(* IEC 61131-3 sources: beckhoffAutomationInterface/ST/Shark/Lib/Communication, 6 files *)

(* ---- GVL_Modbus.st ---- *)
{attribute 'qualified_only'}
(* Modbus protocol constants. *)
VAR_GLOBAL CONSTANT
    MODBUS_MAX_SLAVE_ADDRESS		: BYTE := 247;
    MODBUS_MAX_NETWORK_DEVICES		: BYTE := 8;
    BYTES_PER_REGISTER				: WORD := 2;
    MAX_REGISTERS_PER_OPERATION		: WORD := 32;

    MODBUS_ERROR_INVALID_MASTER		: WORD := 16#8010;
    MODBUS_ERROR_NULL_POINTER		: WORD := 16#8012;
    MODBUS_ERROR_INVALID_QUANTITY	: WORD := 16#8021;
    MODBUS_ERROR_CONVERSION			: WORD := 16#8022;

    MODBUS_DATA_BUFFER_SIZE			: WORD := 64;
    MODBUS_READ_BUFFER_SIZE			: WORD := 32;

    MODBUS_REQUEST_TIMEOUT			: TIME := T#500MS;
END_VAR

(* ---- F_EngineeringToRawCounts.st ---- *)
(* Pure conversion: engineering units to raw Modbus register counts via linear interpolation. *)
FUNCTION F_EngineeringToRawCounts : WORD
VAR_INPUT
    rValue          : LREAL;
    rMinimumValue   : LREAL;
    rFullScale      : LREAL;
    wRawCountsMax   : WORD;
END_VAR
VAR
    rFraction  : LREAL;
    rRawCounts : LREAL;
END_VAR
    IF wRawCountsMax = 0 OR rFullScale <= rMinimumValue THEN
        F_EngineeringToRawCounts := 0;
        RETURN;
    END_IF

    rFraction := (rValue - rMinimumValue) / (rFullScale - rMinimumValue);
    rFraction := LIMIT(0.0, rFraction, 1.0);

    rRawCounts := rFraction * WORD_TO_LREAL(wRawCountsMax);
    F_EngineeringToRawCounts := LREAL_TO_WORD(LIMIT(0.0, rRawCounts, WORD_TO_LREAL(wRawCountsMax)));
END_FUNCTION

(* ---- F_RawCountsToEngineering.st ---- *)
(* Pure conversion: raw Modbus register counts to engineering units via linear interpolation. *)
FUNCTION F_RawCountsToEngineering : LREAL
VAR_INPUT
    wRawCounts      : WORD;
    rMinimumValue   : LREAL;
    rFullScale      : LREAL;
    wRawCountsMax   : WORD;
END_VAR
    IF wRawCountsMax = 0 OR rFullScale <= rMinimumValue THEN
        F_RawCountsToEngineering := 0.0;
        RETURN;
    END_IF

    F_RawCountsToEngineering := rMinimumValue
        + (WORD_TO_LREAL(wRawCounts) / WORD_TO_LREAL(wRawCountsMax))
        * (rFullScale - rMinimumValue);
END_FUNCTION

(* ---- FB_BaseModbusDevice.st ---- *)
(* Base Modbus device handler. Provides FSM for Modbus read/write operations. *)
FUNCTION_BLOCK ABSTRACT FB_BaseModbusDevice IMPLEMENTS I_ModbusSlave
VAR
    _eFSMState 					: E_ModbusDeviceState := E_ModbusDeviceState.IDLE;
    _nUnitId					: BYTE := 0;
    _ipModbusComm				: I_ModbusCommunication := 0;
    _sName						: STRING(80) := 'FB_BaseModbusDevice';
    _fbError					: FB_ErrorHandler;
END_VAR

METHOD PROTECTED SetName
VAR_INPUT
    sName : STRING(80);
END_VAR
    _sName := sName;
    _fbError.Init(sName);
END_METHOD

METHOD PROTECTED RaiseError
VAR_INPUT
    eErrorId : E_ErrorId;
    sMessage : STRING(255);
END_VAR
    _fbError.Raise(eErrorId, sMessage);
END_METHOD

METHOD PROTECTED ClearError
    _fbError.Clear();
END_METHOD

METHOD PUBLIC HandleRequest : BOOL
    IF _eFSMState <> E_ModbusDeviceState.IDLE THEN
        HandleRequest := FALSE;
        RETURN;
    END_IF;

    // NOTE: Do NOT pre-clear the error here. The previous cycle's error stays
    // visible to callers until the next operation actually succeeds, matching
    // the self-healing pattern used by sensors and other controllers.

    // Template-method hook: let the concrete device latch a snapshot of its
    // pending write commands at the start of the transaction. This bounds the
    // write-drain loop even when an upstream controller re-asserts write
    // requests every scan (otherwise the FSM never reaches START_READ/IDLE).
    OnBeginTransaction();

    _eFSMState := E_ModbusDeviceState.START_WRITE;
    HandleRequest := TRUE;
END_METHOD

METHOD PUBLIC Reset : BOOL
    ClearError();
    _eFSMState := E_ModbusDeviceState.IDLE;
    Reset := TRUE;
END_METHOD

METHOD PUBLIC Update : BOOL
    IF _ipModbusComm = 0 THEN
        _eFSMState := E_ModbusDeviceState.IDLE;
        Update := FALSE;
        RETURN;
    END_IF;

    _ipModbusComm.Update();

    CASE _eFSMState OF
        E_ModbusDeviceState.IDLE:
        Update := TRUE;
        RETURN;

        E_ModbusDeviceState.START_WRITE:
        _HandleStartWrite();

        E_ModbusDeviceState.START_READ:
        _HandleStartRead();

        E_ModbusDeviceState.WAIT_FOR_WRITE:
        _HandleWaitForWrite();

        E_ModbusDeviceState.WAIT_FOR_READ:
        _HandleWaitForRead();
    END_CASE;

    Update := TRUE;
END_METHOD

METHOD PRIVATE _HandleStartWrite
VAR
    nWriteStartRegister, nWriteQuantity : WORD;
    pWriteData : POINTER TO BYTE;
END_VAR
    IF GetWritePayload(nStartingRegister => nWriteStartRegister, nQuantity => nWriteQuantity, pData => pWriteData) THEN
        IF _ipModbusComm.StartWriteOperation(nStartRegister := nWriteStartRegister, nQuantity := nWriteQuantity, pData := pWriteData) THEN
            _eFSMState := E_ModbusDeviceState.WAIT_FOR_WRITE;
        END_IF;
    ELSE
        _eFSMState := E_ModbusDeviceState.START_READ;
    END_IF;
END_METHOD

METHOD PRIVATE _HandleStartRead
VAR
    nReadStartRegister, nReadQuantity : WORD;
END_VAR
    IF GetReadPayload(nStartingRegister => nReadStartRegister, nQuantity => nReadQuantity) THEN
        IF _ipModbusComm.StartReadOperation(nStartRegister := nReadStartRegister, nQuantity := nReadQuantity) THEN
            _eFSMState := E_ModbusDeviceState.WAIT_FOR_READ;
        END_IF;
    ELSE
        _eFSMState := E_ModbusDeviceState.IDLE;
    END_IF;
END_METHOD

METHOD PRIVATE _HandleWaitForWrite
VAR
    bSuccess : BOOL;
    wErrorCode : WORD;
END_VAR
    IF NOT _ipModbusComm.IsOperationComplete() THEN
        RETURN;
    END_IF;

    bSuccess := _ipModbusComm.GetOperationResult(wErrorCode);

    IF bSuccess THEN
        ClearError();
        HandleSuccessfulWrite();
    ELSE
        _HandleFailedOperation(wErrorCode);
    END_IF;

    _eFSMState := E_ModbusDeviceState.START_WRITE;
END_METHOD

METHOD PRIVATE _HandleWaitForRead
VAR
    bSuccess : BOOL;
    wErrorCode : WORD;
    pData : POINTER TO BYTE;
    nDataLength : UINT;
END_VAR
    IF NOT _ipModbusComm.IsOperationComplete() THEN
        RETURN;
    END_IF;

    bSuccess := _ipModbusComm.GetOperationResult(wErrorCode);

    IF bSuccess THEN
        ClearError();
        _ipModbusComm.GetReadData(pData, nDataLength);
        HandleSuccessfulRead(pData, nDataLength);
    ELSE
        _HandleFailedOperation(wErrorCode);
    END_IF;

    _eFSMState := E_ModbusDeviceState.IDLE;
END_METHOD

METHOD PRIVATE _HandleFailedOperation
VAR_INPUT
    wErrorCode : WORD;
END_VAR
    RaiseError(E_ErrorId.ERR_COMM_TIMEOUT, CONCAT('Modbus operation failed, code: ', WORD_TO_STRING(wErrorCode)));
END_METHOD

METHOD PUBLIC IsBusy : BOOL
    IsBusy := _eFSMState <> E_ModbusDeviceState.IDLE;
END_METHOD

METHOD PROTECTED _Init : BOOL
VAR_INPUT
    nUnitId						: BYTE;
    ipModbusComm				: I_ModbusCommunication;
END_VAR
    IF ipModbusComm = 0 THEN
        RaiseError(E_ErrorId.ERR_GEN_NULL_POINTER, 'Communication handler is null');
        RETURN;
    END_IF

    _nUnitId := nUnitId;
    _ipModbusComm := ipModbusComm;
    _Init := TRUE;
END_METHOD

METHOD PUBLIC GetUnitId : BYTE
    GetUnitId := _nUnitId;
END_METHOD

METHOD PROTECTED ABSTRACT HandleSuccessfulRead
VAR_INPUT
    pData						: POINTER TO BYTE;
    nDataLength					: UINT;
END_VAR
END_METHOD

METHOD PROTECTED ABSTRACT GetReadPayload : BOOL
VAR_OUTPUT
    nStartingRegister			: WORD;
    nQuantity					: WORD;
END_VAR
END_METHOD

METHOD PROTECTED ABSTRACT GetWritePayload : BOOL
VAR_OUTPUT
    nStartingRegister			: WORD;
    nQuantity					: WORD;
    pData						: POINTER TO BYTE;
END_VAR
END_METHOD

METHOD PROTECTED ABSTRACT HandleSuccessfulWrite
END_METHOD

(* Template-method hook called once at the start of each round-robin transaction
   (IDLE -> START_WRITE). The default implementation is a no-op. Devices whose
   write commands are re-asserted every scan should override this to snapshot the
   pending write requests, so a single transaction stays bounded:
   drain snapshotted writes -> read -> IDLE. *)
METHOD PROTECTED OnBeginTransaction
END_METHOD

END_FUNCTION_BLOCK

(* ---- FB_ModbusHardwareHandler.st ---- *)
(* Modbus hardware communication handler. Wraps Beckhoff ModbusRtuMasterV2_KL6x22B. *)
FUNCTION_BLOCK FB_ModbusHardwareHandler IMPLEMENTS I_ModbusCommunication
VAR
    _fbError            : FB_ErrorHandler;
    _pModbusMaster      : POINTER TO ModbusRtuMasterV2_KL6x22B;
    _nSlaveAddress      : BYTE;
    _bOperationComplete : BOOL := FALSE;
    _wError             : WORD := 0;
    _aDataBuffer        : ARRAY[0..GVL_Modbus.MODBUS_DATA_BUFFER_SIZE-1] OF BYTE;
    _aReadBuffer        : ARRAY[0..GVL_Modbus.MODBUS_READ_BUFFER_SIZE-1] OF WORD;
    _nLastQuantity      : WORD;
    _nLastRegister      : WORD;
    _eLastOperation     : E_ModbusOperationType := E_ModbusOperationType.NONE;
    _bExecuteFlag       : BOOL := FALSE;
END_VAR

METHOD PRIVATE ConvertModbusBytesToWords : BOOL
VAR_INPUT
    pByteData : POINTER TO BYTE;
    nByteCount : WORD;
    pWordBuffer : POINTER TO WORD;
    nMaxWords : WORD;
END_VAR
VAR
    nWordsToConvert : WORD;
END_VAR
    IF pByteData = 0 THEN
        RETURN;
    END_IF

    IF pWordBuffer = 0 THEN
        RETURN;
    END_IF

    IF nByteCount = 0 THEN
        RETURN;
    END_IF

    IF (nByteCount MOD GVL_Modbus.BYTES_PER_REGISTER) <> 0 THEN
        RETURN;
    END_IF

    nWordsToConvert := nByteCount / GVL_Modbus.BYTES_PER_REGISTER;
    IF nWordsToConvert > nMaxWords THEN
        nWordsToConvert := nMaxWords;
    END_IF

    // Bulk copy — data is already in native (little-endian) byte order
    MEMCPY(pWordBuffer, pByteData, nWordsToConvert * SIZEOF(WORD));

    ConvertModbusBytesToWords := TRUE;
END_METHOD

METHOD PRIVATE _ValidateForOperation : BOOL
VAR_INPUT
    nQuantity : WORD;
END_VAR
    IF _pModbusMaster = 0 THEN
        _wError := GVL_Modbus.MODBUS_ERROR_INVALID_MASTER;
        _fbError.Raise(eErrorId := E_ErrorId.ERR_GEN_NULL_POINTER, sMessage := 'Modbus master not initialized');
        RETURN;
    END_IF

    IF _pModbusMaster^.BUSY THEN
        RETURN;
    END_IF

    IF nQuantity = 0 OR nQuantity > GVL_Modbus.MAX_REGISTERS_PER_OPERATION THEN
        _wError := GVL_Modbus.MODBUS_ERROR_INVALID_QUANTITY;
        _fbError.Raise(eErrorId := E_ErrorId.ERR_GEN_INVALID_PARAM, sMessage := 'Invalid register quantity');
        RETURN;
    END_IF

    _ValidateForOperation := TRUE;
END_METHOD

METHOD PUBLIC Init : BOOL
VAR_INPUT
    sInstanceName    : STRING(80);
    pModbusRtuMaster : POINTER TO ModbusRtuMasterV2_KL6x22B;
    nSlaveAddress    : BYTE;
END_VAR
    _fbError.Init(sSourceName := sInstanceName);

    _pModbusMaster := pModbusRtuMaster;
    _nSlaveAddress := nSlaveAddress;

    IF pModbusRtuMaster = 0 THEN
        _fbError.Raise(eErrorId := E_ErrorId.ERR_GEN_NULL_POINTER, sMessage := 'Modbus master pointer is null');
        Init := FALSE;
    ELSE
        _fbError.Clear();
        Init := TRUE;
    END_IF
END_METHOD

METHOD PUBLIC StartReadOperation : BOOL
VAR_INPUT
    nStartRegister : WORD;
    nQuantity : WORD;
END_VAR
    IF NOT _ValidateForOperation(nQuantity := nQuantity) THEN
        RETURN;
    END_IF

    _nLastQuantity := nQuantity;
    _nLastRegister := nStartRegister;
    _eLastOperation := E_ModbusOperationType.READ;
    _bOperationComplete := FALSE;
    _wError := 0;
    _bExecuteFlag := TRUE;
    _fbError.Clear();

    StartReadOperation := TRUE;
END_METHOD

METHOD PUBLIC StartWriteOperation : BOOL
VAR_INPUT
    nStartRegister : WORD;
    nQuantity : WORD;
    pData : POINTER TO BYTE;
END_VAR
    IF NOT _ValidateForOperation(nQuantity := nQuantity) THEN
        RETURN;
    END_IF

    IF pData = 0 THEN
        _wError := GVL_Modbus.MODBUS_ERROR_NULL_POINTER;
        _fbError.Raise(eErrorId := E_ErrorId.ERR_GEN_NULL_POINTER, sMessage := 'Data pointer is null');
        RETURN;
    END_IF

    // Bulk copy — native byte order is little-endian, matching Modbus register layout
    MEMCPY(ADR(_aDataBuffer), pData, nQuantity * GVL_Modbus.BYTES_PER_REGISTER);

    _nLastQuantity := nQuantity;
    _nLastRegister := nStartRegister;
    _eLastOperation := E_ModbusOperationType.WRITE;
    _bOperationComplete := FALSE;
    _wError := 0;
    _bExecuteFlag := TRUE;
    _fbError.Clear();

    StartWriteOperation := TRUE;
END_METHOD

METHOD PUBLIC Update : BOOL
    IF _pModbusMaster = 0 THEN
        _bOperationComplete := TRUE;
        _wError := GVL_Modbus.MODBUS_ERROR_INVALID_MASTER;
        _fbError.Raise(eErrorId := E_ErrorId.ERR_GEN_NULL_POINTER, sMessage := 'Modbus master not initialized');
        Update := TRUE;
        RETURN;
    END_IF

    IF _eLastOperation = E_ModbusOperationType.NONE THEN
        Update := _bOperationComplete;
        RETURN;
    END_IF

    _CallMaster();

    IF NOT _bOperationComplete AND_THEN NOT _pModbusMaster^.BUSY THEN
        _bOperationComplete := TRUE;
        _HandleCompletion();
        _eLastOperation := E_ModbusOperationType.NONE;
    END_IF

    Update := _bOperationComplete;
END_METHOD

METHOD PRIVATE _CallMaster
VAR
    nByteLength : WORD;
END_VAR
    nByteLength := _nLastQuantity * GVL_Modbus.BYTES_PER_REGISTER;

    IF _eLastOperation = E_ModbusOperationType.READ THEN
        _pModbusMaster^.ReadRegs(
            UnitID := _nSlaveAddress,
            Quantity := _nLastQuantity,
            MBAddr := _nLastRegister,
            cbLength := nByteLength,
            pMemoryAddr := ADR(_aDataBuffer),
            Execute := _bExecuteFlag,
            Timeout := GVL_Modbus.MODBUS_REQUEST_TIMEOUT
        );
    ELSIF _eLastOperation = E_ModbusOperationType.WRITE THEN
        _pModbusMaster^.WriteRegs(
            UnitID := _nSlaveAddress,
            Quantity := _nLastQuantity,
            MBAddr := _nLastRegister,
            cbLength := nByteLength,
            pMemoryAddr := ADR(_aDataBuffer),
            Execute := _bExecuteFlag,
            Timeout := GVL_Modbus.MODBUS_REQUEST_TIMEOUT
        );
    END_IF

    _bExecuteFlag := FALSE;
END_METHOD

METHOD PRIVATE _HandleCompletion
VAR
    nActualBytes : WORD;
END_VAR
    IF _pModbusMaster^.Error THEN
        _wError := INT_TO_WORD(_pModbusMaster^.ErrorId);
        _fbError.Raise(eErrorId := E_ErrorId.ERR_COMM_PROTOCOL,
            sMessage := CONCAT('Modbus error code: ', WORD_TO_STRING(_wError)));
        RETURN;
    END_IF

    IF _eLastOperation <> E_ModbusOperationType.READ THEN
        RETURN;
    END_IF

    nActualBytes := UDINT_TO_WORD(_pModbusMaster^.cbRead);

    IF nActualBytes = 0 THEN
        _wError := GVL_Modbus.MODBUS_ERROR_CONVERSION;
        _fbError.Raise(eErrorId := E_ErrorId.ERR_COMM_INVALID_RESPONSE, sMessage := 'No data received');
    ELSIF nActualBytes > GVL_Modbus.MODBUS_DATA_BUFFER_SIZE THEN
        _wError := GVL_Modbus.MODBUS_ERROR_CONVERSION;
        _fbError.Raise(eErrorId := E_ErrorId.ERR_COMM_BUFFER_OVERFLOW, sMessage := 'Response exceeds buffer size');
    ELSIF NOT ConvertModbusBytesToWords(
        pByteData := ADR(_aDataBuffer),
        nByteCount := nActualBytes,
        pWordBuffer := ADR(_aReadBuffer),
        nMaxWords := GVL_Modbus.MODBUS_READ_BUFFER_SIZE
    ) THEN
        _wError := GVL_Modbus.MODBUS_ERROR_CONVERSION;
        _fbError.Raise(eErrorId := E_ErrorId.ERR_COMM_DATA_CONVERSION, sMessage := 'Byte to word conversion failed');
    END_IF
END_METHOD

METHOD PUBLIC IsOperationComplete : BOOL
    IsOperationComplete := _bOperationComplete;
END_METHOD

METHOD PUBLIC GetOperationResult : BOOL
VAR_INPUT
    wErrorCode : REFERENCE TO WORD;
END_VAR
    wErrorCode := _wError;
    GetOperationResult := (_wError = 0);
END_METHOD

METHOD PUBLIC GetReadData : BOOL
VAR_INPUT
    pData : REFERENCE TO POINTER TO BYTE;
    nDataLength : REFERENCE TO UINT;
END_VAR
    pData := ADR(_aReadBuffer);
    nDataLength := WORD_TO_UINT(_nLastQuantity * GVL_Modbus.BYTES_PER_REGISTER);
    GetReadData := TRUE;
END_METHOD

METHOD PUBLIC GetSlaveAddress : BYTE
    GetSlaveAddress := _nSlaveAddress;
END_METHOD

END_FUNCTION_BLOCK

(* ---- FB_ModbusNetworkCoordinator.st ---- *)
(* Modbus network coordinator. Round-robin scheduler for shared-bus Modbus slaves. *)
FUNCTION_BLOCK FB_ModbusNetworkCoordinator
VAR_OUTPUT
    nCurrentSlaveIndex : BYTE := 0;
END_VAR
VAR
    _aSlaves : ARRAY[1..GVL_Modbus.MODBUS_MAX_NETWORK_DEVICES] OF I_ModbusSlave;
    _ipActiveSlave : I_ModbusSlave;
    _tonNetworkSettling : TON;
    _tSettlingTime : TIME := T#5MS;
    _eNetworkState : E_NetworkState := E_NetworkState.SELECT_SLAVE;
    _nNumSlaves : BYTE := 0;
    _bInitialized : BOOL := FALSE;
END_VAR

VAR CONSTANT
    MIN_SLAVE_INDEX : BYTE := 1;
END_VAR

METHOD PUBLIC AddSlave : BOOL
VAR_INPUT
    ipSlave : I_ModbusSlave;
END_VAR
VAR
    i : BYTE;
END_VAR
    IF ipSlave = 0 THEN
        RETURN;
    END_IF

    IF _nNumSlaves >= GVL_Modbus.MODBUS_MAX_NETWORK_DEVICES THEN
        RETURN;
    END_IF

    FOR i := 1 TO _nNumSlaves DO
        IF _aSlaves[i] = ipSlave THEN
            RETURN;
        END_IF
    END_FOR

    _nNumSlaves := _nNumSlaves + 1;
    _aSlaves[_nNumSlaves] := ipSlave;
    AddSlave := TRUE;
END_METHOD

METHOD PUBLIC Init : BOOL
VAR_INPUT
    tSettlingTime : TIME := T#5MS;
END_VAR
    IF _nNumSlaves = 0 THEN
        RETURN;
    END_IF

    _tSettlingTime := tSettlingTime;
    nCurrentSlaveIndex := MIN_SLAVE_INDEX;
    _eNetworkState := E_NetworkState.SELECT_SLAVE;
    _tonNetworkSettling(IN := FALSE);
    _ipActiveSlave := 0;
    _bInitialized := TRUE;
    Init := TRUE;
END_METHOD

METHOD PUBLIC Execute : BOOL
    IF NOT _bInitialized THEN
        RETURN;
    END_IF

    CASE _eNetworkState OF
        E_NetworkState.SELECT_SLAVE:
            IF nCurrentSlaveIndex = 0 OR nCurrentSlaveIndex > _nNumSlaves THEN
                nCurrentSlaveIndex := MIN_SLAVE_INDEX;
            END_IF
            _ipActiveSlave := _aSlaves[nCurrentSlaveIndex];
            _eNetworkState := E_NetworkState.INITIATE_REQUEST;

        E_NetworkState.INITIATE_REQUEST:
            IF _ipActiveSlave <> 0 AND_THEN NOT _ipActiveSlave.IsBusy() THEN
                _ipActiveSlave.HandleRequest();
                _eNetworkState := E_NetworkState.AWAIT_COMPLETION;
            ELSE
                _eNetworkState := E_NetworkState.SETTLING;
                _tonNetworkSettling(IN := TRUE, PT := _tSettlingTime);
            END_IF

        E_NetworkState.AWAIT_COMPLETION:
            IF _ipActiveSlave <> 0 THEN
                _ipActiveSlave.Update();
                IF NOT _ipActiveSlave.IsBusy() THEN
                    _eNetworkState := E_NetworkState.SETTLING;
                    _tonNetworkSettling(IN := TRUE, PT := _tSettlingTime);
                END_IF
            ELSE
                _eNetworkState := E_NetworkState.SETTLING;
                _tonNetworkSettling(IN := TRUE, PT := _tSettlingTime);
            END_IF

        E_NetworkState.SETTLING:
            _tonNetworkSettling();
            IF _tonNetworkSettling.Q THEN
                _tonNetworkSettling(IN := FALSE);
                _ipActiveSlave := 0;
                nCurrentSlaveIndex := (nCurrentSlaveIndex MOD _nNumSlaves) + 1;
                _eNetworkState := E_NetworkState.SELECT_SLAVE;
            END_IF
    END_CASE

    Execute := TRUE;
END_METHOD

METHOD PUBLIC GetSlaveCount : BYTE
    GetSlaveCount := _nNumSlaves;
END_METHOD

METHOD PUBLIC GetNetworkState : E_NetworkState
    GetNetworkState := _eNetworkState;
END_METHOD

END_FUNCTION_BLOCK
